TYPE "UDT_ZC_DISP_PPAL_PID"
VERSION : 0.1
   STRUCT
      Orden : Bool;   // Orden activacion
      Consigna : Real;   // Consigna
      ValorActual : Real;   // Valor actual
   END_STRUCT;

END_TYPE

